{attribute 'linkalways'} 
{attribute 'no_explicit_call' := 'This FB is a CLASS and must be accessed using methods or properties'}
{attribute 'enable_dynamic_creation'}
FUNCTION_BLOCK FINAL SEL_LREAL EXTENDS Node
VAR
	g : _BOOL(FALSE);
	in1 : _LREAL(0.0);
	in2 : _LREAL(0.0);
	out : _LREAL(0.0);
END_VAR

METHOD PUBLIC Clone : I_Node
VAR
	pNode : POINTER TO SEL_LREAL;
END_VAR
pNode := __NEW(SEL_LREAL);
Clone := pNode^;
END_METHOD

METHOD FB_init : BOOL
VAR_INPUT
	bInitRetains : BOOL; // if TRUE, the retain variables are initialized (warm start / cold start)
	bInCopyCode : BOOL;  // if TRUE, the instance afterwards gets moved into the copy code (online change)
END_VAR
AddInput('g',THIS^.g);
AddInput('in1',THIS^.in1);
AddInput('in2',THIS^.in2);
AddOutput('out', THIS^.out);
END_METHOD

METHOD PROTECTED OnExecute
VAR
END_VAR
IF g.value THEN
	out.value := in2.value;
ELSE
	out.value := in1.value;
END_IF
END_METHOD

END_FUNCTION_BLOCK

(* stored: Version 1.1.0.1, ProductVersion 3.1.4024.15
   POU SEL_LREAL: Id {99b5f450-dd27-44cd-819b-4801f7d1c9dd}, SpecialFunc None
   Folder Constructor: Id {e5af1280-81b5-4912-ab00-6f1410d9ae52}
   Method Clone: Id {c5382658-21cb-47aa-a69a-9607a63b2c85}
   Method FB_init: Id {9f518609-3180-4760-9e58-f12c7dabc540}
   Method OnExecute: Id {6fc05581-9876-450f-be91-8682d92d6566} *)
